{attribute 'linkalways'} 
{attribute 'no_explicit_call' := 'This FB is a CLASS and must be accessed using methods or properties'}
{attribute 'enable_dynamic_creation'}
FUNCTION_BLOCK Node_F_VN_ConvertCartesianToPolarAnglesExp EXTENDS VisionNode
VAR
	ipSrcPointsCart : _ITcVnContainer;
    ipDestAngles : _ITcVnContainer;
    bAngleInDegrees : _BOOL(FALSE);
    hrPrev : _HRESULT(S_OK);
	hresult : _HRESULT(S_OK);
END_VAR

METHOD PUBLIC  Clone : I_Node
VAR
	pNode : POINTER TO Node_F_VN_ConvertCartesianToPolarAnglesExp;
END_VAR
pNode := __NEW(Node_F_VN_ConvertCartesianToPolarAnglesExp);
Clone := pNode^;
END_METHOD

METHOD FB_init : BOOL
VAR_INPUT
	bInitRetains : BOOL; // if TRUE, the retain variables are initialized (warm start / cold start)
	bInCopyCode : BOOL;  // if TRUE, the instance afterwards gets moved into the copy code (online change)
END_VAR
AddInput('ipSrcPointsCart', ipSrcPointsCart);
AddParameter('bAngleInDegrees', bAngleInDegrees);
AddInput('hrPrev', hrPrev);
AddOutput('ipDestAngles', ipDestAngles);
AddOutput('hresult',hresult);
END_METHOD

METHOD PROTECTED OnExecute
hresult.Value := F_VN_ConvertCartesianToPolarAnglesExp(
	ipSrcPointsCart := ipSrcPointsCart.Value,
	ipDestAngles := ipDestAngles.Value,
    bAngleInDegrees := bAngleInDegrees.Value,
	hrPrev := hrPrev.Value);
END_METHOD

METHOD PUBLIC PreExecutionCheck
VAR_INPUT
	Check : I_PreExecutionChecks;
END_VAR
Check.IsTrue(ipSrcPointsCart.IsValid, 'ipSrcPointsCart must be a valid container');
Check.IsTrue((ipSrcPointsCart.IsType(TC_GLOBAL_CONST_LIST.ContainerType_Vector_TcVnPoint2_DINT) OR
              ipSrcPointsCart.IsType(TC_GLOBAL_CONST_LIST.ContainerType_Vector_TcVnPoint2_REAL) OR
              ipSrcPointsCart.IsType(TC_GLOBAL_CONST_LIST.ContainerType_Vector_TcVnPoint2_LREAL)),
              'ipSrcPointsCart contains incorrect type');
END_METHOD

END_FUNCTION_BLOCK

(* stored: Version 1.1.0.1, ProductVersion 3.1.4026.13
   POU Node_F_VN_ConvertCartesianToPolarAnglesExp: Id {405e209e-6fa1-0345-1be1-61bb5088a5ab}, SpecialFunc None
   Folder Constructor: Id {daea2751-c5e7-06d1-29e3-21ceaf4288fa}
   Method Clone: Id {cc5b87bf-6c67-06dd-3ca6-b77444f1467e}
   Method FB_init: Id {bd29c243-cc09-03f7-3d9c-70011481137d}
   Method OnExecute: Id {691a69ef-b2ed-0147-0c5d-b1afafecd781}
   Method PreExecutionCheck: Id {a0eb7e1b-e593-0df6-2e38-4c9330254b2c} *)
